// TIA Portal V17 export
// export: Created 2021-12-03T08:08:04.7602753Z, ExportSetting WithDefaults, DisplayName Totally Integrated Automation Portal, DisplayVersion V17, DisplayName TIA Portal Openness, DisplayVersion V17, DisplayName TIA Portal Version Control Interface, DisplayVersion V17, DisplayName STEP 7 Professional, DisplayVersion V17, DisplayName STEP 7 Safety, DisplayVersion V17, DisplayName WinCC Advanced, DisplayVersion V17
VAR_GLOBAL   // PLC tag table "Digital_Inputs"
   I_BrLigSrvFlt AT %I0.0 : Bool;   // Breaker Light and Service Outlet Fault
   I_BrModFlt AT %I0.1 : Bool;   // Breaker Modulator Fault
   I_BrChilFlt AT %I0.2 : Bool;   // Breaker Chiller Fault
   I_BrPow1Flt AT %I0.3 : Bool;   // Breaker Powersupply 1 24VDC Fault
   I_BrPow2Flt AT %I0.4 : Bool;   // Breaker Powersupply 2 24VDC Fault
   I_BrFrqConvFlt AT %I0.5 : Bool;   // Breaker Frequnce Converter Conveyor Fault
   I_BrAccConFlt AT %I0.6 : Bool;   // Breaker Accelerator Console Fault
   I_BrXRayUnitFlt AT %I0.7 : Bool;   // Breaker X-Ray Unit Fault
   I_BrPowPlcFlt AT %I1.0 : Bool;   // Breaker Powersupply PS307 (PLC) Fault
   I_SitopPow1Flt AT %I1.1 : Bool;   // Sitop Diagnose Modul Powersupply 1 Failure
   I_SitopPow2Flt AT %I1.2 : Bool;   // Sitop Diagnose Modul Powersupply 2 Failure
   I_BrMod1PFlt AT %I1.3 : Bool;   // Breaker Modulator 230 VAC Fault
   I_P2ConvLocal AT %I3.0 : Bool;   // Panel 2: Keyswitch Conveyor Local
   "I_/P2ConvLocal" AT %I3.1 : Bool;   // Panel 2: Keyswitch Conveyor Local (False=Local)
   I_P2ConvFwd AT %I3.2 : Bool;   // Panel 2: Conveyor move forward
   I_P2ConvBwd AT %I3.3 : Bool;   // Panel 2: Conveyor move backward
   I_AccStRemMode AT %I4.0 : Bool;   // Accelerator Status: Remote Mode selected
   I_AccStPowerOn AT %I4.1 : Bool;   // Accelerator Status: Power on
   I_AccStWarmUp AT %I4.2 : Bool;   // Accelerator Status: Warming up
   I_AccStClear AT %I4.3 : Bool;   // Accelerator Status: Clear
   I_AccStReady AT %I4.4 : Bool;   // Accelerator Status: Ready
   I_AccStXRayOn AT %I4.5 : Bool;   // Accelerator Status: X-Ray on
   I_AccStFault AT %I4.6 : Bool;   // Accelerator Status: Fault
   I_AccStNoEmStp AT %I4.7 : Bool;   // Accelerator Status: Emergency Stop not active
   I_PSConvStpBwd AT %I5.0 : Bool;   // Photo Sensor Conveyor Stop Position Back
   I_PSConvSlowBwd AT %I5.1 : Bool;   // Photo Sensor Conveyor Fast Slow Back
   I_PSConvSlowFwd AT %I5.2 : Bool;   // Photo Sensor Conveyor Fast Slow Front
   I_PSConvStpFwd AT %I5.3 : Bool;   // Photo Sensor Conveyor Stop Position Front
   I_PSConvXRayBwd AT %I5.4 : Bool;   // Photo Sensor Conveyor Sensor X-Ray Back
   I_PSConvXRayFwd AT %I5.5 : Bool;   // Photo Sensor Conveyor Sensor X-Ray Front
   I_Spare5_6 AT %I5.6 : Bool;   // Spare
   I_Spare5_7 AT %I5.7 : Bool;   // Spare
   I_ChilVlv_Acc1_Pos AT %I6.0 : Bool;   // Chiller Valve Position 1
   I_ChilVlv_Acc2_Pos AT %I6.1 : Bool;   // Chiller Valve Position 2
   I_ModSwch_Acc1_Pos AT %I6.2 : Bool;   // Modulator Switch Position 1
   I_ModSwch_Acc2_Pos AT %I6.3 : Bool;   // Modulator Switch Position 2
   I_Spare6_4 AT %I6.4 : Bool;   // Spare
   I_Spare6_5 AT %I6.5 : Bool;   // Spare
   I_Spare6_6 AT %I6.6 : Bool;   // Spare
   I_Spare6_7 AT %I6.7 : Bool;   // Spare
   I_AccStStandby AT %I7.0 : Bool;   // Accelerator Status: Standby
   I_AccStMicroWave AT %I7.1 : Bool;   // Accelerator Status: Microwave (TIS, MIS)
   I_AccStHighDoze AT %I7.2 : Bool;   // Accelerator Status: High Doze (MIS)
   I_AccStRemouteKey AT %I7.3 : Bool;   // Accelerator Status: Acc Panel Key
   I_AccStEmStpPanel AT %I7.4 : Bool;   // Accelerator Status: Emergency Stop Panel (True=No EmStp)
   I_Spare1_4 AT %I1.4 : Bool;   // Spare
   I_Spare1_5 AT %I1.5 : Bool;   // Spare
   I_Spare1_6 AT %I1.6 : Bool;   // Spare
   I_Spare1_7 AT %I1.7 : Bool;   // Spare
   I_Spare2_0 AT %I2.0 : Bool;   // Spare
   I_Spare2_1 AT %I2.1 : Bool;   // Spare
   I_Spare2_2 AT %I2.2 : Bool;   // Spare
   I_Spare2_3 AT %I2.3 : Bool;   // Spare
   I_Spare2_4 AT %I2.4 : Bool;   // Spare
   I_Spare2_5 AT %I2.5 : Bool;   // Spare
   I_Spare2_6 AT %I2.6 : Bool;   // Spare
   I_Spare2_7 AT %I2.7 : Bool;   // Spare
   I_Spare3_4 AT %I3.4 : Bool;   // Spare
   I_Spare3_5 AT %I3.5 : Bool;   // Spare
   I_Spare3_6 AT %I3.6 : Bool;   // Spare
   I_Spare3_7 AT %I3.7 : Bool;   // Spare
   I_Spare7_5 AT %I7.5 : Bool;   // Spare
   I_Spare7_6 AT %I7.6 : Bool;   // Spare
   I_Spare7_7 AT %I7.7 : Bool;   // Spare
END_VAR
